# EPICS substitutions: old/bl6-SkfChopper/bl6-SkfChopperApp/Db/skf4_ioc_sns.substitutions
file ioc_sns.db
{
pattern {IOCNAME}
        {BL6:IocSts:ChopSkf4}
}
